(* CODESYS project hello_plc_application.export

Project tree, tasks and I/O mapping:
  application hello_plc_application
    task MainTask (cyclic, interval 200 ms, priority 30, watchdog 20 ms x 1) calls PLC_PRG
    program PLC_PRG [ST]
    Symbols
*)

// hello_plc_application/PLC_PRG
{attribute 'symbol' := 'readwrite'}

PROGRAM PLC_PRG
VAR

	strVar01	:	STRING(255):='Empty string #1';
	strVar02	:	STRING(255):='Empty string #2';
	
	rVar01		:	REAL:=0.0;
	rVar02		:	REAL:=0.0;
	
	iVar01		:	INT:=0;
	iVar02		:	INT:=0;
END_VAR

// Dummy code to avoid warnings
IF (strVar01 <> strVar02) THEN
	; 
END_IF

IF (rVar01 <> rVar02) THEN
	;
END_IF

IF (iVar01 <> iVar02) THEN
	;
END_IF

END_PROGRAM
